RoboDK station: Lab03_TovarOspina.rdk

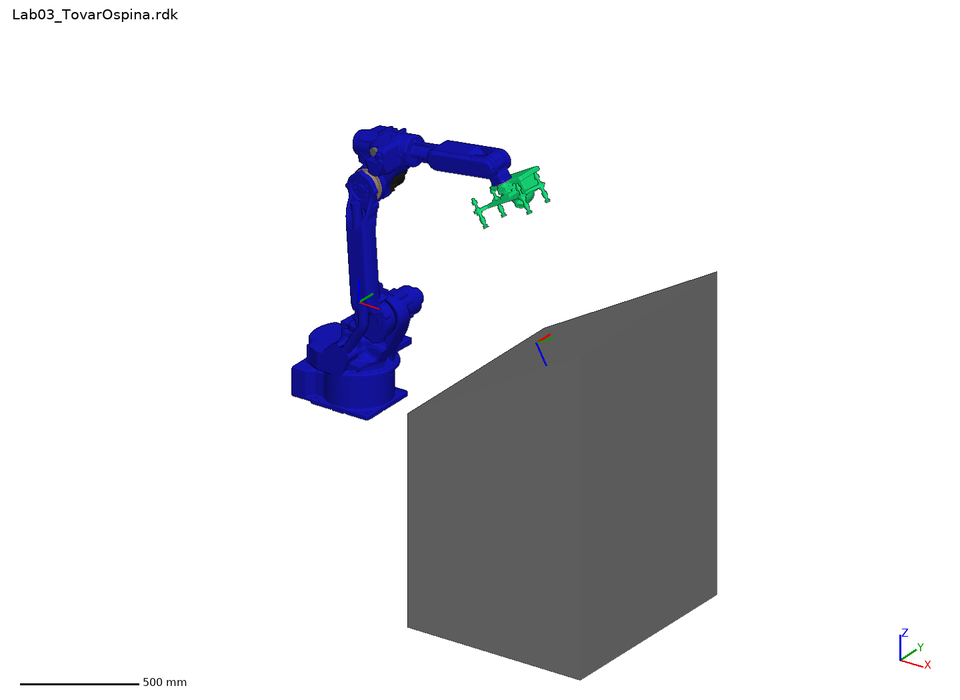
[picture v0: the station drawn from its stored meshes, robots at their saved joint values, targets as dots, program paths as lines]
Station Robodk (2) (saved by RoboDK 5.9.1). Poses are relative to the parent item; angles as X-Y-Z fixed-axis rotations.
  - frame Motoman MH6 Base at (0, 0, 450) mm
    - robot Motoman MH6: 6 axes, payload 6 kg, reach 1422 mm, repeatability 0.08 mm, weight 130 kg
        modified DH rows (alpha deg, a mm, theta deg, d mm): 0, 0, 0, 450; -90, 152, -90, 0; 0, 614, 0, 0; -90, 155, 0, 640; 90, 0, 90, 0; -90, 0, 0, 95
        base shift (0, 0, -450) mm
        joint limits [-170, -90, -175, -180, -45, -360] to [170, 155, 250, 180, 225, 360]; home [0, 0, 0, 0, 0, 0]; saved at [-2.758, -4.034, 4.933, -1.477, 20.998, 92.918]
      - tool Ventosas, TCP at (0, 0, 190) mm, size 250 x 290 x 148 mm
    - frame Frame_from_Target1 at (935.29, -34.49, 85.5) mm, rotated rx 150 ry 0 rz 90 deg
  - object CAJA2 at (1600, 500, 300) mm, rotated rx 180 ry 0 rz 0 deg, size 886.4 x 1000 x 1511.7 mm, geometry from CAJA2.stp
  - Python program RosPolar (listed below)

--- Python program RosPolar ---
from robodk.robolink import *    # API para comunicarte con RoboDK
from robodk.robomath import *    # Funciones matemáticas
import math

#------------------------------------------------
# 1) Conexión a RoboDK e inicialización
#------------------------------------------------
RDK = Robolink()

# Elegir un robot (si hay varios, aparece un popup)
robot = RDK.ItemUserPick("Selecciona un robot", ITEM_TYPE_ROBOT)
if not robot.Valid():
    raise Exception("No se ha seleccionado un robot válido.")

# Conectar al robot físico
##if not robot.Connect():
##    raise Exception("No se pudo conectar al robot. Verifica que esté en modo remoto y que la configuración sea correcta.")
##
### Confirmar conexión
##if not robot.ConnectedState():
##    raise Exception("El robot no está conectado correctamente. Revisa la conexión.")
##
##print("Robot conectado correctamente.")

#------------------------------------------------
# 2) Cargar el Frame (ya existente) donde quieres dibujar
#    Ajusta el nombre si tu Frame se llama diferente
#------------------------------------------------
frame_name = "Frame_from_Target1"
frame = RDK.Item(frame_name, ITEM_TYPE_FRAME)
if not frame.Valid():
    raise Exception(f'No se encontró el Frame "{frame_name}" en la estación.')

# Asignamos este frame al robot
robot.setPoseFrame(frame)
# Usamos la herramienta activa
robot.setPoseTool(robot.PoseTool())

# Ajustes de velocidad y blending
robot.setSpeed(300)   # mm/s - Ajusta según necesites
robot.setRounding(5)  # blending (radio de curvatura)

#------------------------------------------------
# 3) Parámetros de la figura (rosa polar)
#------------------------------------------------
num_points = 920       # Cuántos puntos muestreamos (mayor = más suave)
A = 150               # Amplitud (300 mm = radio máximo)
k = 5/2                  # Parámetro de la rosa (pétalos). Si es impar, habrá k pétalos; si es par, 2k
z_surface = 0          # Z=0 en el plano del frame
z_safe = 50            # Altura segura para aproximarse y salir

#------------------------------------------------
# 4) Movimiento al centro en altura segura
#------------------------------------------------
# El centro de la rosa (r=0) corresponde a x=0, y=0
robot.MoveJ(transl(0, 200, -500))

robot.MoveJ(transl(0, 0, z_surface + z_safe))

# Bajamos a la "superficie" (Z=0)
robot.MoveL(transl(0, 0, z_surface))

#------------------------------------------------
# 5) Dibujar la rosa polar
#    r = A * sin(k*theta)
#    x = r*cos(theta), y = r*sin(theta)
#------------------------------------------------
# Recorremos theta de 0 a 2*pi (una vuelta completa)
full_turn = 4*math.pi

for i in range(num_points+1):
    # Fracción entre 0 y 1
    t = i / num_points
    # Ángulo actual
    theta = full_turn * t

    # Calculamos r
    r = A * math.sin(k * theta)

    # Convertimos a coordenadas Cartesianas X, Y
    x = r * math.cos(theta)
    y = r * math.sin(theta)

    # Movemos linealmente (MoveL) en el plano del Frame
    robot.MoveJ(transl(x, y, z_surface))

robot.MoveJ(transl(0, 200, -500))

robot.MoveL(transl(0, 400, z_surface))
robot.MoveL(transl(0, 200, z_surface))
robot.MoveL(transl(100, 200, z_surface))
robot.MoveL(transl(100, 250, z_surface))
robot.MoveL(transl(100, 250, z_surface - z_safe))

robot.MoveL(transl(-200, 400, z_surface - z_safe))
robot.MoveL(transl(-200, 400, z_surface))
robot.MoveL(transl(-100, 400, z_surface))
robot.MoveL(transl(-100, 300, z_surface))
robot.MoveL(transl(-200, 300, z_surface))
robot.MoveL(transl(-200, 200, z_surface))
robot.MoveL(transl(-100, 200, z_surface))



# Al terminar, subimos de nuevo para no chocar
robot.MoveL(transl(x, y, z_surface + z_safe))

robot.MoveJ(transl(0, 200, -500))

print(f"¡Figura (rosa polar) completada en el frame '{frame_name}'!")
